_CFC_ (* Continuous Function Chart, elements in execution order *)
#0 RT_VKL_OLD_SEZ_LETO:R_TRIG(CLK: TRUE)
#1 MOVE(EN: #0.Q, 20)
#2 SHU6_PV1_UST_SEZ_LETO_OLD <= #1
#3 RT_VKL_OLD_SEZ_ZIMA:R_TRIG(CLK: TRUE)
#4 MOVE(EN: #3.Q, 19)
#5 SHU6_PV1_UST_SEZ_ZIMA_OLD <= #4
#6 <>(SHU6_PV1_UST_SEZ_LETO, SHU6_PV1_UST_SEZ_LETO_OLD)
#7 >(SHU6_PV1_UST_SEZ_LETO, SHU6_PV1_UST_SEZ_ZIMA_OLD)
#8 AND(#6, #7)
#9 MOVE(EN: #8, SHU6_PV1_UST_SEZ_LETO)
#10 SHU6_PV1_UST_SEZ_LETO_OLD <= #9
#11 AND(#6, NOT #7)
#12 MOVE(EN: #11, SHU6_PV1_UST_SEZ_LETO_OLD)
#13 SHU6_PV1_UST_SEZ_LETO <= #12
#14 <>(SHU6_PV1_UST_SEZ_ZIMA, SHU6_PV1_UST_SEZ_LETO_OLD)
#15 <(SHU6_PV1_UST_SEZ_ZIMA, SHU6_PV1_UST_SEZ_LETO_OLD)
#16 AND(#14, #15)
#17 MOVE(EN: #16, SHU6_PV1_UST_SEZ_ZIMA)
#18 SHU6_PV1_UST_SEZ_ZIMA_OLD <= #17
#19 AND(#14, NOT #15)
#20 MOVE(EN: #19, SHU6_PV1_UST_SEZ_ZIMA_OLD)
#21 SHU6_PV1_UST_SEZ_ZIMA <= #20
#22 RT_TE6_UST_OTKL_OLD:R_TRIG(CLK: TRUE)
#23 MOVE(EN: #22.Q, 22)
#24 SHU6_PV1_TE6_UST_OTKL_OLD <= #23
#25 RT_TE6_UST_VKL_OLD:R_TRIG(CLK: TRUE)
#26 MOVE(EN: #25.Q, 19)
#27 SHU6_PV1_TE6_UST_VKL_OLD <= #26
#28 <>(SHU6_PV1_TE6_UST_OTKL, SHU6_PV1_TE6_UST_OTKL_OLD)
#29 >(SHU6_PV1_TE6_UST_OTKL, SHU6_PV1_TE6_UST_VKL_OLD)
#30 AND(#28, #29)
#31 MOVE(EN: #30, SHU6_PV1_TE6_UST_OTKL)
#32 SHU6_PV1_TE6_UST_OTKL_OLD <= #31
#33 AND(#28, NOT #29)
#34 MOVE(EN: #33, SHU6_PV1_TE6_UST_OTKL_OLD)
#35 SHU6_PV1_TE6_UST_OTKL <= #34
#36 <>(SHU6_P1_1_TE6_UST_VKL, SHU6_PV1_TE6_UST_VKL_OLD)
#37 <(SHU6_P1_1_TE6_UST_VKL, SHU6_PV1_TE6_UST_OTKL_OLD)
#38 AND(#36, #37)
#39 MOVE(EN: #38, SHU6_P1_1_TE6_UST_VKL)
#40 SHU6_PV1_TE6_UST_VKL_OLD <= #39
#41 AND(#36, NOT #37)
#42 MOVE(EN: #41, SHU6_PV1_TE6_UST_VKL_OLD)
#43 SHU6_P1_1_TE6_UST_VKL <= #42
_END_CFC_
END_PROGRAM

(* POU Input/AI/TE1, CFC *)
PROGRAM TE1
VAR
	fb_TE1: ISTOK_ANALOGVH;
	ofset: REAL;
	fb_SHU6_PV1_TE1_B_UST_MYAG_REG: ISTOK_GT;
	fb_SHU6_PV1_TE1_B_UST_SEZ_LETO: ISTOK_GT;
	I_GT_TE: ISTOK_GT;
	I_LT_TE: ISTOK_LT;
	TON_DOST: TON;
END_VAR
VAR (* helpers for the ST form of the networks *)
	_t94 : BOOL;
	_t75 : REAL;
END_VAR
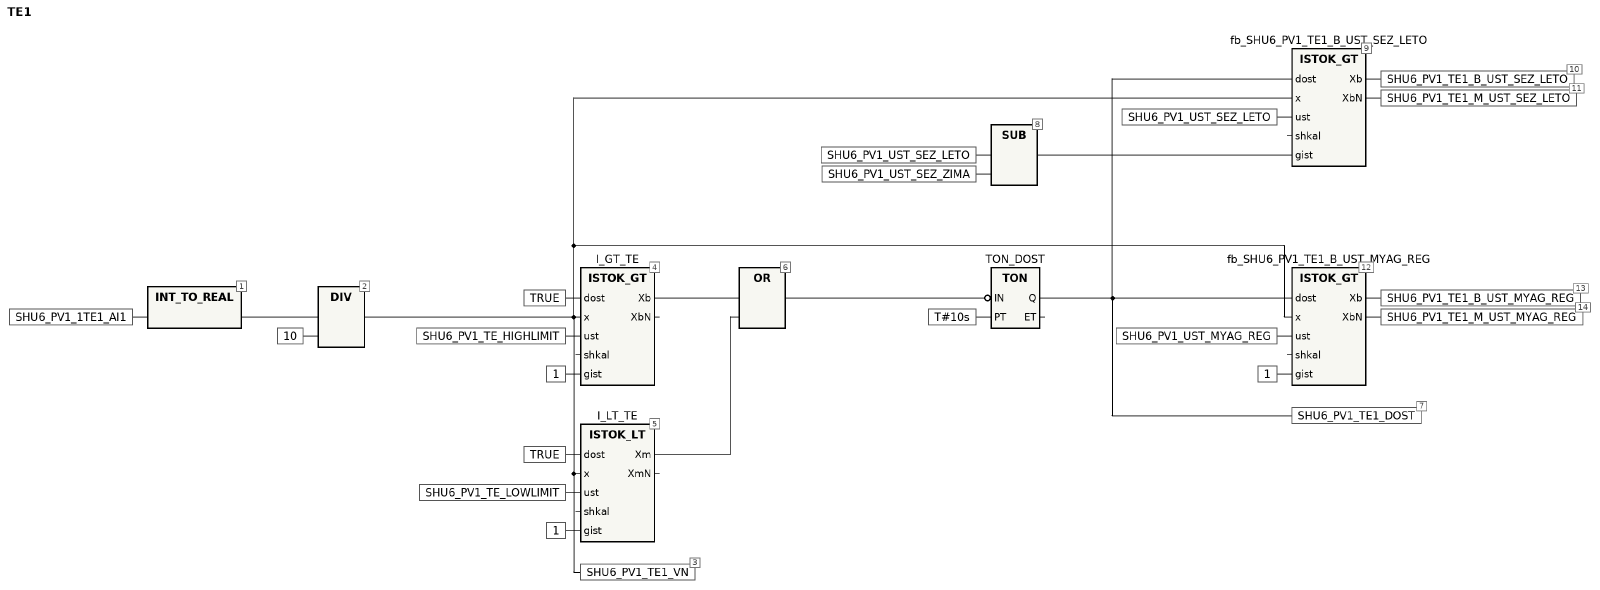
